(* IEC 61131-3 sources: horner-cscape-mcp/artifacts/projects/FailAudit_POU_UndeclaredVariable/pous, 1 file *)

(* ---- POU_UndeclaredVariable.st ---- *)
PROGRAM POU_UndeclaredVariable
VAR
    ValidLevel : REAL := 25.0;
END_VAR
UnallocatedSensor := 99.9;
END_PROGRAM
